(* CoDeSys 2.3 export: WORK.EXP *)

(* POU workHour, LD *)
PROGRAM workHour
VAR
	evlev1_hour : calcHOUR;
	CONV_1_hour : calcHOUR;
	FAN_1_hour : calcHOUR;
	MILL_1_hour : calcHOUR;
	SEP_1_hour : calcHOUR;
	CONV_2_hour : calcHOUR;
	FAN_2_hour : calcHOUR;

	MILL_2_hour: calcHOUR;
	SEP_2_hour: calcHOUR;
	SHNEK_1_hour: calcHOUR;
	SHNEK_2_hour: calcHOUR;
	STAR_11_hour: calcHOUR;
	STAR_12_hour: calcHOUR;
	STAR_21_hour: calcHOUR;
	STAR_22_hour: calcHOUR;
	OIL_1_hour: calcHOUR;
	OIL_2_hour: calcHOUR;
	SHNK_SIKL_1_hour: calcHOUR;
	SHNK_SIKL_2_hour: calcHOUR;

END_VAR
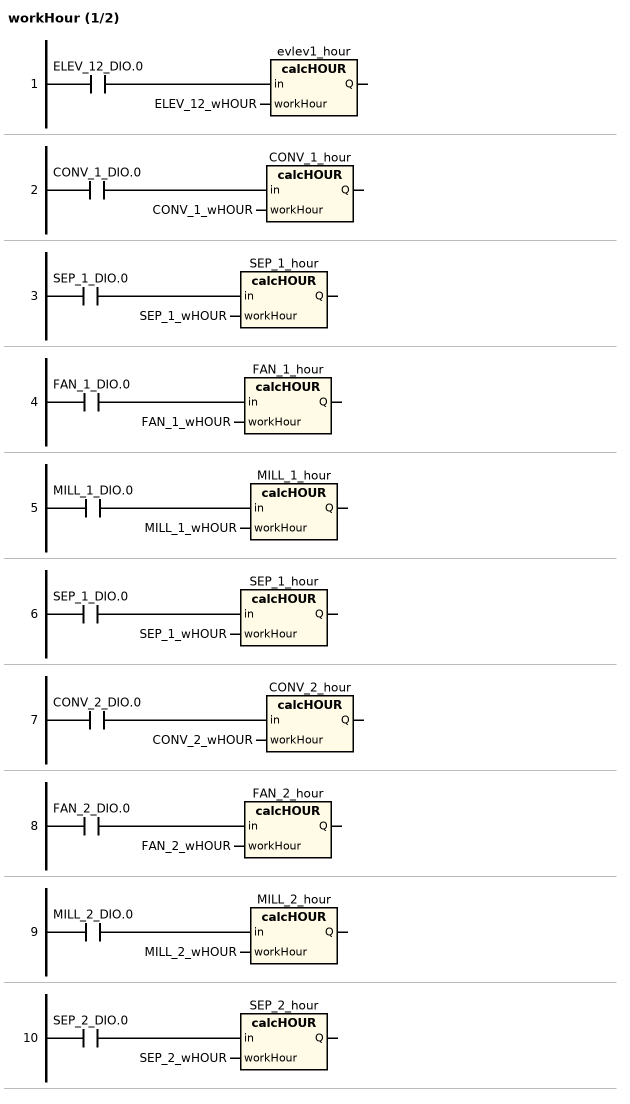
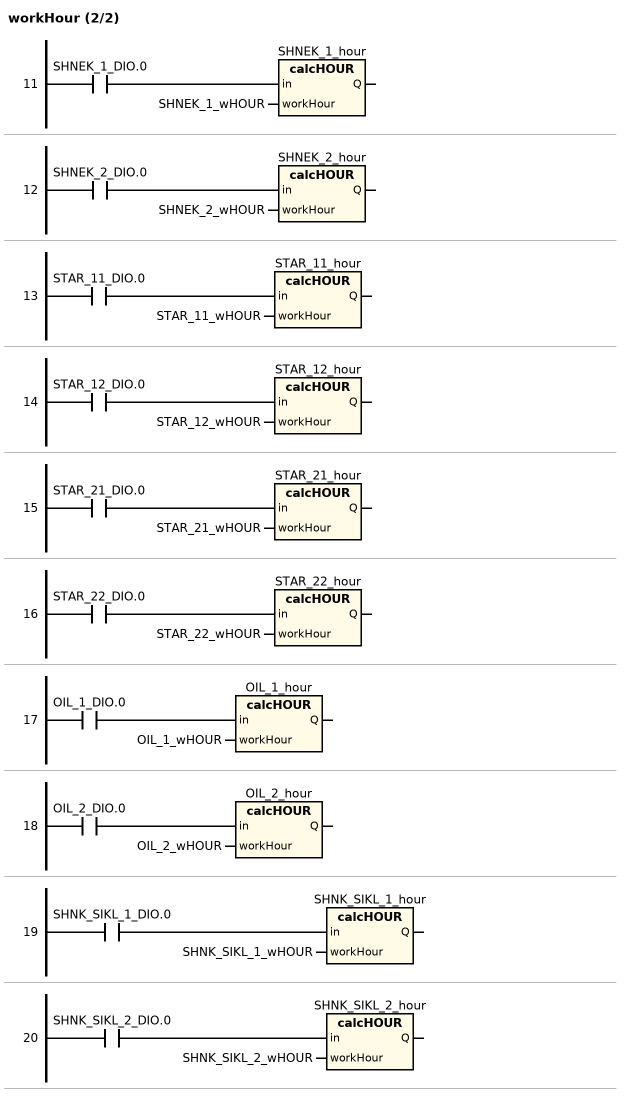
_LD_ (* Ladder Diagram *)
NETWORK 1
	[ELEV_12_DIO.0] - evlev1_hour:calcHOUR(in: *, workHour: ELEV_12_wHOUR)
NETWORK 2
	[CONV_1_DIO.0] - CONV_1_hour:calcHOUR(in: *, workHour: CONV_1_wHOUR)
NETWORK 3
	[SEP_1_DIO.0] - SEP_1_hour:calcHOUR(in: *, workHour: SEP_1_wHOUR)
NETWORK 4
	[FAN_1_DIO.0] - FAN_1_hour:calcHOUR(in: *, workHour: FAN_1_wHOUR)
NETWORK 5
	[MILL_1_DIO.0] - MILL_1_hour:calcHOUR(in: *, workHour: MILL_1_wHOUR)
NETWORK 6
	[SEP_1_DIO.0] - SEP_1_hour:calcHOUR(in: *, workHour: SEP_1_wHOUR)
NETWORK 7
	[CONV_2_DIO.0] - CONV_2_hour:calcHOUR(in: *, workHour: CONV_2_wHOUR)
NETWORK 8
	[FAN_2_DIO.0] - FAN_2_hour:calcHOUR(in: *, workHour: FAN_2_wHOUR)
NETWORK 9
	[MILL_2_DIO.0] - MILL_2_hour:calcHOUR(in: *, workHour: MILL_2_wHOUR)
NETWORK 10
	[SEP_2_DIO.0] - SEP_2_hour:calcHOUR(in: *, workHour: SEP_2_wHOUR)
NETWORK 11
	[SHNEK_1_DIO.0] - SHNEK_1_hour:calcHOUR(in: *, workHour: SHNEK_1_wHOUR)
NETWORK 12
	[SHNEK_2_DIO.0] - SHNEK_2_hour:calcHOUR(in: *, workHour: SHNEK_2_wHOUR)
NETWORK 13
	[STAR_11_DIO.0] - STAR_11_hour:calcHOUR(in: *, workHour: STAR_11_wHOUR)
NETWORK 14
	[STAR_12_DIO.0] - STAR_12_hour:calcHOUR(in: *, workHour: STAR_12_wHOUR)
NETWORK 15
	[STAR_21_DIO.0] - STAR_21_hour:calcHOUR(in: *, workHour: STAR_21_wHOUR)
NETWORK 16
	[STAR_22_DIO.0] - STAR_22_hour:calcHOUR(in: *, workHour: STAR_22_wHOUR)
NETWORK 17
	[OIL_1_DIO.0] - OIL_1_hour:calcHOUR(in: *, workHour: OIL_1_wHOUR)
NETWORK 18
	[OIL_2_DIO.0] - OIL_2_hour:calcHOUR(in: *, workHour: OIL_2_wHOUR)
NETWORK 19
	[SHNK_SIKL_1_DIO.0] - SHNK_SIKL_1_hour:calcHOUR(in: *, workHour: SHNK_SIKL_1_wHOUR)
NETWORK 20
	[SHNK_SIKL_2_DIO.0] - SHNK_SIKL_2_hour:calcHOUR(in: *, workHour: SHNK_SIKL_2_wHOUR)
_END_LD_
(* the same logic as Structured Text *)
(* Network 1 *)
evlev1_hour(in := ELEV_12_DIO.0, workHour := ELEV_12_wHOUR);
(* Network 2 *)
CONV_1_hour(in := CONV_1_DIO.0, workHour := CONV_1_wHOUR);
(* Network 3 *)
SEP_1_hour(in := SEP_1_DIO.0, workHour := SEP_1_wHOUR);
(* Network 4 *)
FAN_1_hour(in := FAN_1_DIO.0, workHour := FAN_1_wHOUR);
(* Network 5 *)
MILL_1_hour(in := MILL_1_DIO.0, workHour := MILL_1_wHOUR);
(* Network 6 *)
SEP_1_hour(in := SEP_1_DIO.0, workHour := SEP_1_wHOUR);
(* Network 7 *)
CONV_2_hour(in := CONV_2_DIO.0, workHour := CONV_2_wHOUR);
(* Network 8 *)
FAN_2_hour(in := FAN_2_DIO.0, workHour := FAN_2_wHOUR);
(* Network 9 *)
MILL_2_hour(in := MILL_2_DIO.0, workHour := MILL_2_wHOUR);
(* Network 10 *)
SEP_2_hour(in := SEP_2_DIO.0, workHour := SEP_2_wHOUR);
(* Network 11 *)
SHNEK_1_hour(in := SHNEK_1_DIO.0, workHour := SHNEK_1_wHOUR);
(* Network 12 *)
SHNEK_2_hour(in := SHNEK_2_DIO.0, workHour := SHNEK_2_wHOUR);
(* Network 13 *)
STAR_11_hour(in := STAR_11_DIO.0, workHour := STAR_11_wHOUR);
(* Network 14 *)
STAR_12_hour(in := STAR_12_DIO.0, workHour := STAR_12_wHOUR);
(* Network 15 *)
STAR_21_hour(in := STAR_21_DIO.0, workHour := STAR_21_wHOUR);
(* Network 16 *)
STAR_22_hour(in := STAR_22_DIO.0, workHour := STAR_22_wHOUR);
(* Network 17 *)
OIL_1_hour(in := OIL_1_DIO.0, workHour := OIL_1_wHOUR);
(* Network 18 *)
OIL_2_hour(in := OIL_2_DIO.0, workHour := OIL_2_wHOUR);
(* Network 19 *)
SHNK_SIKL_1_hour(in := SHNK_SIKL_1_DIO.0, workHour := SHNK_SIKL_1_wHOUR);
(* Network 20 *)
SHNK_SIKL_2_hour(in := SHNK_SIKL_2_DIO.0, workHour := SHNK_SIKL_2_wHOUR);
END_PROGRAM

(* POU calcHOUR, CFC *)
FUNCTION_BLOCK calcHOUR
VAR_INPUT
	in : BOOL;
END_VAR
VAR_IN_OUT
	workHour : WORD;
END_VAR
VAR
	tp1: TP;
	go : BOOL;
	rtrig: R_TRIG;
	ctu1: CTU;
	vaqt : WORD := 3600;
END_VAR
VAR (* helpers for the ST form of the networks *)
	_t14 : WORD;
	_en14 : BOOL;
END_VAR
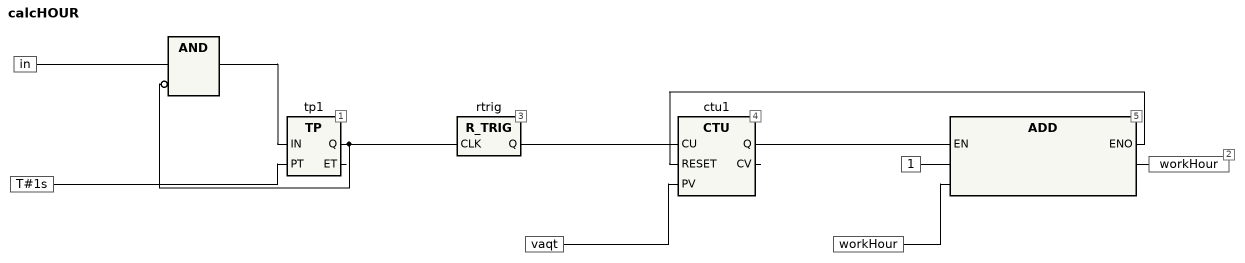
_CFC_ (* Continuous Function Chart, elements in execution order *)
#0 AND(in, NOT #1.Q)
#1 tp1:TP(IN: #0, PT: T#1s)
#2 workHour <= #5
#3 rtrig:R_TRIG(CLK: #1.Q)
#4 ctu1:CTU(CU: #3.Q, RESET: #5.ENO, PV: vaqt)
#5 ADD(EN: #4.Q, 1, workHour)
_END_CFC_
(* the same logic as Structured Text *)
tp1(IN := in AND NOT tp1.Q, PT := T#1s);
workHour := _t14;
rtrig(CLK := tp1.Q);
ctu1(CU := rtrig.Q, RESET := _en14, PV := vaqt);
_en14 := ctu1.Q;
IF _en14 THEN _t14 := 1 + workHour; END_IF;
END_FUNCTION_BLOCK
